FUNCTION_BLOCK INTERNAL FINAL FB_ReadRepeatedFieldFixed64Tests EXTENDS FB_TestSuite
VAR_INPUT
END_VAR
VAR_OUTPUT
END_VAR
VAR
	aActual             : ARRAY [0..7] OF LINT;
    fbFieldCodec 		: FB_FieldCodecFixed64(nTag:= 16#0A);
	fbRepeatedField		: FB_RepeatedField(anyArray:= F_ToAnyType(aActual), anyFirstElem:= F_ToAnyType(aActual[0]), ipFieldCodec:= fbFieldCodec);
END_VAR

ShouldReadRepeatedFieldTheory();

METHOD PRIVATE Reset
VAR_INPUT
END_VAR
fbRepeatedField.Initialize();
MEMSET(destAddr:= ADR(aActual), fillByte:= 16#0, n:= SIZEOF(aActual));
END_METHOD

METHOD PRIVATE ShouldReadRepeatedField
VAR_IN_OUT CONSTANT
    aBuffer     : ARRAY [*] OF BYTE;
    aExpected   : ARRAY [*] OF LINT;
END_VAR
VAR_INPUT CONSTANT
    nBufferPosStart     : UDINT;
    nExpectedBufferPos  : UDINT;
    nExpectedFieldIndex : UDINT;
    ipFieldCodec        : I_FieldCodec;
END_VAR
VAR_INST
    fbCtx               : FB_ParseContext;
END_VAR
VAR
    hr                  : HRESULT;
    nTag                : UDINT;
END_VAR
// Arrange
Reset();
fbCtx.FromBuffer(aBuffer);
fbCtx.refCtx.stState.nBufferPos := nBufferPosStart;

// Act
F_ParseTag(fbCtx.refCtx, nTag=> nTag);
hr := fbRepeatedField.AddEntriesFrom(fbParseCtx:= fbCtx, ipFieldCodec:= ipFieldCodec);

// Assert
AssertEquals_DINT(
    Expected:= S_OK,
    Actual:= hr,
    Message:= 'Expected S_OK instead of error');
    
{warning disable C0041}
AssertArrayEquals_LINT(Expecteds:= aExpected, Actuals:= aActual, Message:= '');
 
AssertEquals_UDINT(
    Expected:= nExpectedBufferPos,
    Actual:= fbCtx.refCtx.stState.nBufferPos,
    Message:= CONCAT('Expected stState.nBufferPos to equal ', TO_STRING(nExpectedBufferPos)));
    
AssertEquals_UDINT(
    Expected:= nExpectedFieldIndex,
    Actual:= fbRepeatedField.nCount,
    Message:= CONCAT('Expected fbRepeatedField.nCount to equal ', TO_STRING(nExpectedFieldIndex)));
END_METHOD

METHOD PRIVATE ShouldReadRepeatedFieldTheory : REFERENCE TO FB_Test
(*
    syntax = "proto3";
    
    message exampleMessage
    {
      repeated fixed32 repeatedFixed32 = 4;
    }
*)
VAR CONSTANT
    cRawValueZeroLength     : ARRAY[0..31] OF BYTE := [16#22, 16#00];       // field #4
    cRawValue1              : ARRAY[0..100] OF BYTE := [16#22, 16#30, 16#00, 16#00, 16#00, 16#00, 16#00, 16#00, 16#00, 16#00, 16#d2, 16#04, 16#00, 16#00, 16#00, 16#00, 16#00, 16#00, 16#39, 16#05, 16#00, 16#00, 16#00, 16#00, 16#00, 16#00, 16#ff, 16#ff, 16#ff, 16#ff, 16#ff, 16#ff, 16#ff, 16#ff, 16#c7, 16#fa, 16#ff, 16#ff, 16#ff, 16#ff, 16#ff, 16#ff, 16#4e, 16#61, 16#bc, 16#00, 16#00, 16#00, 16#00, 16#00];
    
END_VAR

VAR CONSTANT
    aExpectedZeroLength     : ARRAY [0..7] OF LINT := [0, 0, 0, 0, 0, 0, 0, 0];
    aExpected1              : ARRAY [0..7] OF LINT := [0, 1234, 1337, -1, -1337, 12345678, 0, 0];
END_VAR
TEST(__POUNAME());

ShouldReadRepeatedField(aBuffer:= cRawValueZeroLength, aExpected:= aExpectedZeroLength, nBufferPosStart:= 0, nExpectedBufferPos:= 2, nExpectedFieldIndex:= 0, ipFieldCodec:= THIS^.fbFieldCodec);
ShouldReadRepeatedField(aBuffer:= cRawValue1, aExpected:= aExpected1, nBufferPosStart:= 0, nExpectedBufferPos:= 50, nExpectedFieldIndex:= 6, ipFieldCodec:= THIS^.fbFieldCodec);

TEST_FINISHED_NAMED(__POUNAME());
END_METHOD

END_FUNCTION_BLOCK

(* stored: Version 1.1.0.1
   POU FB_ReadRepeatedFieldFixed64Tests: Id {2f2a1335-1f41-4851-a210-cf1bdd05c323}, SpecialFunc None
   Method Reset: Id {ebca8802-1d89-41f4-8f9f-5bd3dc41475c}
   Method ShouldReadRepeatedField: Id {e5bc7800-7458-4f36-ba28-c5a97662bd36}
   Method ShouldReadRepeatedFieldTheory: Id {cc58d154-3c36-4882-9cd2-1709d6eeb781} *)
